// TIA Portal V21 export
FUNCTION "Main trends" : Void   // FC31, LAD
{ S7_Optimized_Access := 'TRUE' }
// stored: SetENOAutomatically false
BEGIN

REGION Network 1: Gestione trend 1
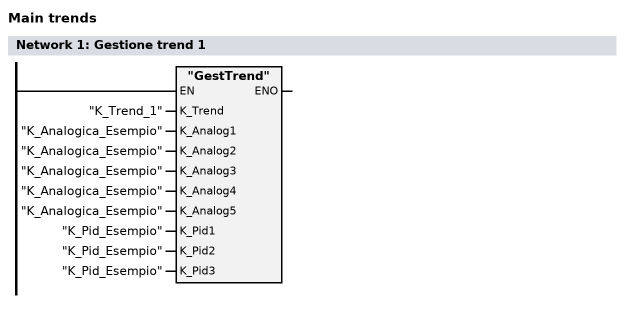
   RUNG wire#powerrail
      "GestTrend"(K_Trend := "K_Trend_1", K_Analog1 := "K_Analogica_Esempio", K_Analog2 := "K_Analogica_Esempio", K_Analog3 := "K_Analogica_Esempio", K_Analog4 := "K_Analogica_Esempio", K_Analog5 := "K_Analogica_Esempio", K_Pid1 := "K_Pid_Esempio", K_Pid2 := "K_Pid_Esempio", K_Pid3 := "K_Pid_Esempio")
   END_RUNG
   // the same network as SCL:
   "GestTrend"(K_Trend := "K_Trend_1",
               K_Analog1 := "K_Analogica_Esempio",
               K_Analog2 := "K_Analogica_Esempio",
               K_Analog3 := "K_Analogica_Esempio",
               K_Analog4 := "K_Analogica_Esempio",
               K_Analog5 := "K_Analogica_Esempio",
               K_Pid1 := "K_Pid_Esempio",
               K_Pid2 := "K_Pid_Esempio",
               K_Pid3 := "K_Pid_Esempio");
END_REGION
END_FUNCTION
